// TIA Portal V20 export
// export: Created 2025-12-01T14:57:24.1996615Z, ExportSetting None, DisplayName Totally Integrated Automation Portal, DisplayVersion V20 Update 3, DisplayName TIA Portal Openness, DisplayVersion V20 Update 3, DisplayName TIA Portal Version Control Interface, DisplayVersion V20 Update 3, DisplayName STEP 7 Professional, DisplayVersion V20 Update 3, DisplayName STEP 7 Safety, DisplayVersion V20 Update 2, DisplayName WinCC Basic/Comfort/Advanced, DisplayVersion V20 Update 3, DisplayName WinCC Professional, DisplayVersion V20 Update 3, DisplayName WinCC Unified, DisplayVersion V20 Update 3
FUNCTION "FC961_ScadaMaquina" : Void   // FC961, STL
TITLE = Funcion de Tratamiento de la Mesa para el SCADA
{ S7_Optimized_Access := 'FALSE' }
AUTHOR : SCADA
NAME : 20161001
VERSION : 1.0
// stored: AutoNumber false
   VAR_INPUT
      NumMaquina : UInt;
   END_VAR
   VAR_TEMP
      Maquina : UInt;
      EnError : Bool;
      EnMarcha : Bool;
   END_VAR
BEGIN

NETWORK
TITLE = Inicializacion
//////////////////////////////////////////////////////////////////////////////
//////////////////////////////////////////////////////////////////////////////
/// Tareas Iniciales de Inicializacion

      L     #NumMaquina;  // Numero de Maquina a tratar
      T     #Maquina;



NETWORK
TITLE = Contadores de Flujos
//////////////////////////////////////////////////////////////////////////////
//////////////////////////////////////////////////////////////////////////////
/// Calculo de Bultos de Entrada

/// -- Bultos de Operacion 01
      SET;
      A     "DB012_ScadaMaquinas".Maquina[#Maquina].Orden_OP1;  // Operacion
      FP    "DB012_ScadaMaquinas".Maquina[#Maquina].MemoBultos_OP1;
      JCN   NBO1;  // Una entrada mas ?

      L     "DB012_ScadaMaquinas".Maquina[#Maquina].Bultos_OP1;  // +1
      L     1;
      +I;
      T     "DB012_ScadaMaquinas".Maquina[#Maquina].Bultos_OP1;

NBO1: NOP   0;


/// -- Bultos de Operacion 02
      SET;
      A     "DB012_ScadaMaquinas".Maquina[#Maquina].Orden_OP2;  // Operacion
      FP    "DB012_ScadaMaquinas".Maquina[#Maquina].MemoBultos_OP2;
      JCN   NBO2;  // Una entrada mas ?

      L     "DB012_ScadaMaquinas".Maquina[#Maquina].Bultos_OP2;  // +1
      L     1;
      +I;
      T     "DB012_ScadaMaquinas".Maquina[#Maquina].Bultos_OP2;

NBO2: NOP   0;

/// -- Bultos de Operacion 03
      SET;
      A     "DB012_ScadaMaquinas".Maquina[#Maquina].Orden_OP3;  // Operacion
      FP    "DB012_ScadaMaquinas".Maquina[#Maquina].MemoBultos_OP3;
      JCN   NBO3;  // Una entrada mas ?

      L     "DB012_ScadaMaquinas".Maquina[#Maquina].Bultos_OP3;  // +1
      L     1;
      +I;
      T     "DB012_ScadaMaquinas".Maquina[#Maquina].Bultos_OP3;

NBO3: NOP   0;

/// -- Bultos de Operacion 04
      SET;
      A     "DB012_ScadaMaquinas".Maquina[#Maquina].Orden_OP4;  // Operacion
      FP    "DB012_ScadaMaquinas".Maquina[#Maquina].MemoBultos_OP4;
      JCN   NBO4;  // Una entrada mas ?

      L     "DB012_ScadaMaquinas".Maquina[#Maquina].Bultos_OP4;  // +1
      L     1;
      +I;
      T     "DB012_ScadaMaquinas".Maquina[#Maquina].Bultos_OP4;

NBO4: NOP   0;

/// -- Bultos de Operacion 01
      SET;
      A     "DB012_ScadaMaquinas".Maquina[#Maquina].Orden_OP5;  // Operacion
      FP    "DB012_ScadaMaquinas".Maquina[#Maquina].MemoBultos_OP5;
      JCN   NBO5;  // Una entrada mas ?

      L     "DB012_ScadaMaquinas".Maquina[#Maquina].Bultos_OP5;  // +1
      L     1;
      +I;
      T     "DB012_ScadaMaquinas".Maquina[#Maquina].Bultos_OP5;

NBO5: NOP   0;



NETWORK
TITLE = Tiempo de Fallo
//////////////////////////////////////////////////////////////////////////////
//////////////////////////////////////////////////////////////////////////////
/// Calculo de Tiempo

      SET;  // En Error
      A     "DB904_Estado_Maquinas".EstadoVI[#Maquina].Error_MAQx;
      =     #EnError;

      SET;
      AN    #EnError;  // Contar Tiempo ?
      JC    N_ER;

      CALL  "FC914_SumaTiempo_DT"
      ( TiempoActual := "DB012_ScadaMaquinas".Maquina[#Maquina].TMP_Error
      );

N_ER: NOP   0;



NETWORK
TITLE = Informacion de los Motores
//////////////////////////////////////////////////////////////////////////////
//////////////////////////////////////////////////////////////////////////////
/// Calculo de Arranques

/// ---- Numero de Arranques del M1 // Subir y Bajar Elevacion
      SET;
      A     "DB904_Estado_Maquinas".EstadoVI[#Maquina].Byte10_bit0;
      O     "DB904_Estado_Maquinas".EstadoVI[#Maquina].Byte10_bit1;
      FP    "DB012_ScadaMaquinas".Maquina[#Maquina].MemoArranques_M1;
      JCN   NAM1;  // Un arranque Mas mas ?

      L     "DB012_ScadaMaquinas".Maquina[#Maquina].Arranques_M1;  // +1
      L     1;
      +I;
      T     "DB012_ScadaMaquinas".Maquina[#Maquina].Arranques_M1;

NAM1: NOP   0;


/// -- Numero de Arranques del M2 // Horq Dch y Izq
      SET;
      A     "DB904_Estado_Maquinas".EstadoVI[#Maquina].Byte10_bit2;
      O     "DB904_Estado_Maquinas".EstadoVI[#Maquina].Byte10_bit3;
      O     "DB904_Estado_Maquinas".EstadoVI[#Maquina].Byte10_bit4;
      O     "DB904_Estado_Maquinas".EstadoVI[#Maquina].Byte10_bit5;
      FP    "DB012_ScadaMaquinas".Maquina[#Maquina].MemoArranques_M2;
      JCN   NAM2;  // Un arranque Mas mas ?

      L     "DB012_ScadaMaquinas".Maquina[#Maquina].Arranques_M2;  // +1
      L     1;
      +I;
      T     "DB012_ScadaMaquinas".Maquina[#Maquina].Arranques_M2;

NAM2: NOP   0;


/// -- Numero de Arranques del M3 // Motor Futuro
      SET;
      A     "DB904_Estado_Maquinas".EstadoVI[#Maquina].Byte11_bit0;
      O     "DB904_Estado_Maquinas".EstadoVI[#Maquina].Byte11_bit1;
      FP    "DB012_ScadaMaquinas".Maquina[#Maquina].MemoArranques_M3;
      JCN   NAM3;  // Un arranque Mas mas ?

      L     "DB012_ScadaMaquinas".Maquina[#Maquina].Arranques_M3;  // +1
      L     1;
      +I;
      T     "DB012_ScadaMaquinas".Maquina[#Maquina].Arranques_M3;

NAM3: NOP   0;





NETWORK
TITLE = ---
//////////////////////////////////////////////////////////////////////////////
//////////////////////////////////////////////////////////////////////////////
/// Calculo de Tiempo

/// -- Tiempo en Marcha M1 // Subir y Bajar Elevacion
      SET;
      A     "DB904_Estado_Maquinas".EstadoVI[#Maquina].Byte10_bit0;
      O     "DB904_Estado_Maquinas".EstadoVI[#Maquina].Byte10_bit1;
      =     #EnMarcha;

      AN    #EnMarcha;  // Contar Tiempo ?
      JC    N_M1;

      CALL  "FC914_SumaTiempo_DT"
      ( TiempoActual := "DB012_ScadaMaquinas".Maquina[#Maquina].TMP_Marcha_M1
      );

N_M1: NOP   0;



// ---- Tiempo en Marcha M2 // Horq Dch y Izq
      SET;
      A     "DB904_Estado_Maquinas".EstadoVI[#Maquina].Byte10_bit2;
      O     "DB904_Estado_Maquinas".EstadoVI[#Maquina].Byte10_bit3;
      O     "DB904_Estado_Maquinas".EstadoVI[#Maquina].Byte10_bit4;
      O     "DB904_Estado_Maquinas".EstadoVI[#Maquina].Byte10_bit5;
      =     #EnMarcha;

      AN    #EnMarcha;  // Contar Tiempo ?
      JC    N_M2;

      CALL  "FC914_SumaTiempo_DT"
      ( TiempoActual := "DB012_ScadaMaquinas".Maquina[#Maquina].TMP_Marcha_M2
      );

N_M2: NOP   0;



// ---- Tiempo en Marcha M3 // Motor Futuro
      SET;
      A     "DB904_Estado_Maquinas".EstadoVI[#Maquina].Byte11_bit0;
      O     "DB904_Estado_Maquinas".EstadoVI[#Maquina].Byte11_bit1;
      =     #EnMarcha;

      AN    #EnMarcha;  // Contar Tiempo ?
      JC    N_M3;

      CALL  "FC914_SumaTiempo_DT"
      ( TiempoActual := "DB012_ScadaMaquinas".Maquina[#Maquina].TMP_Marcha_M3
      );

N_M3: NOP   0;



NETWORK
TITLE = Final de la Funcion
//////////////////////////////////////////////////////////////////////////////
//////////////////////////////////////////////////////////////////////////////
/// Tareas de Finalizacion de la Funcion


END_FUNCTION
